TYPE ST_EmptyServiceParam :
STRUCT
	bDummyValue : BOOL;	// To avoid 0 size check error during Service Coordinator Registration
END_STRUCT
END_TYPE

(* stored: Version 1.1.0.1, ProductVersion 3.1.4026.18
   DUT ST_EmptyServiceParam: Id {c3dc3c66-babe-4b14-814e-557c86aa89f9} *)
